FUNCTION_BLOCK FB_MotionClearAsserts
(*
    Clear all of the PMPS asserts related to a states mover.
*)
VAR_IN_OUT
    // All states to deactivate
    astDbStateParams: ARRAY[*] OF ST_DbStateParams;
    // The arbiter who made the PMPS assert requests
    fbArbiter: FB_ARBITER;
END_VAR
VAR_INPUT
    // Clear asserts on rising edge
    bExecute: BOOL;
END_VAR
VAR_OUTPUT
END_VAR
VAR
    rtExec: R_TRIG;
    nIter: DINT;
END_VAR


rtExec(CLK:=bExecute);
IF rtExec.Q THEN
    FOR nIter := LOWER_BOUND(astDbStateParams, 1) TO UPPER_BOUND(astDbStateParams, 1) DO
        fbArbiter.RemoveRequest(astDbStateParams[nIter].nRequestAssertionID);
    END_FOR
END_IF

END_FUNCTION_BLOCK

(* stored: Version 1.1.0.1, ProductVersion 3.1.4022.18
   POU FB_MotionClearAsserts: Id {26ecf392-a1f3-491b-ac84-9ace07a64d4f}, SpecialFunc None *)
